// TwinCAT 3 PLC project PLC101
// ProgramVersion: 3.1.4022.3
// libraries:
//   Tc2_Standard, * (Beckhoff Automation GmbH)
//   Tc2_System, * (Beckhoff Automation GmbH)
//   Tc3_Module, * (Beckhoff Automation GmbH)
//   TcUnit, * (www.tcunit.org)
// project tree:
//   / PlcTask.TcTTO
//   POUs/ MAIN.TcPOU, FB_TcUnitSuite.TcPOU

CONFIGURATION PLC101
    RESOURCE PLC ON TwinCAT3
        TASK PlcTask(INTERVAL := T#10ms, PRIORITY := 20);
        PROGRAM MAIN WITH PlcTask : MAIN;
    END_RESOURCE
END_CONFIGURATION

// ---- POUs/MAIN.TcPOU
PROGRAM MAIN
VAR
    fbTestSuite : FB_TcUnitSuite;
END_VAR

TcUnit.RUN();

END_PROGRAM

// ---- POUs/FB_TcUnitSuite.TcPOU
{attribute 'call_after_init'}
FUNCTION_BLOCK FB_TcUnitSuite EXTENDS FB_TestSuite
VAR_INPUT
END_VAR
VAR_OUTPUT
END_VAR
VAR
END_VAR

FailingTest();

METHOD FailingTest
VAR_INPUT
END_VAR
TEST('FailingTest');

AssertTrue( FALSE, 'This test always fails');

TEST_FINISHED();
END_METHOD

END_FUNCTION_BLOCK
